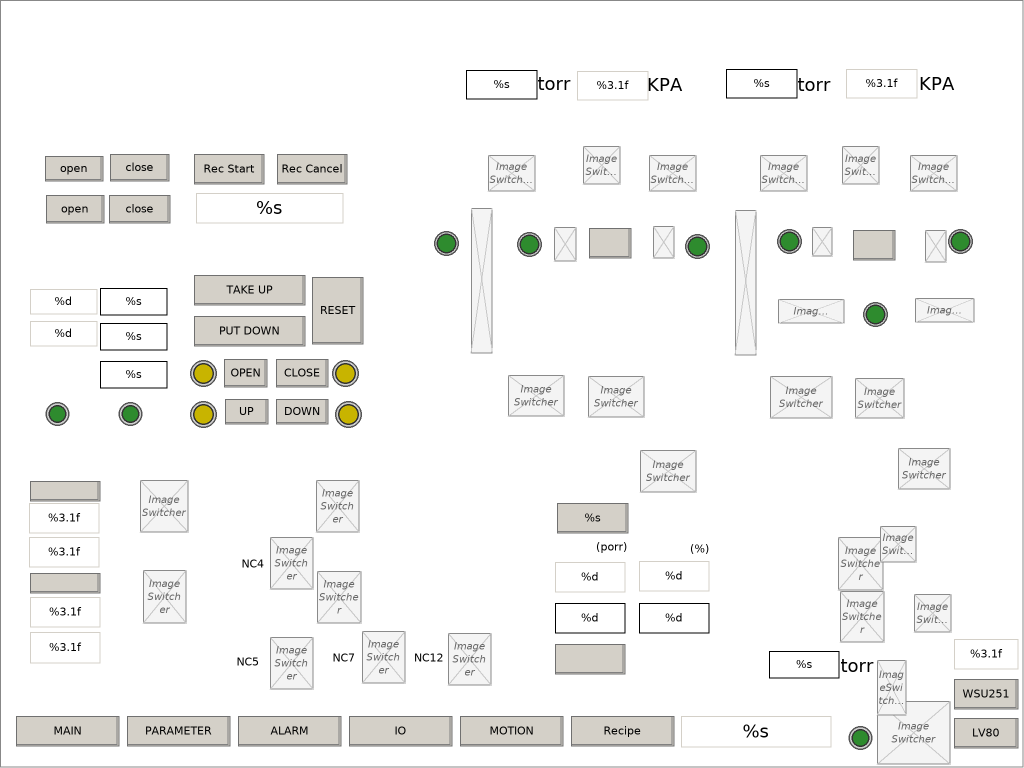
VISUALIZATION MainBase  // 1024x768, background image ImagePool_Base.LAYOUT
    ImageSwitcher (140,480 48x52), variable: DO2_0, background image: ImagePool_Base.VAL_ON, image: ImagePool_Base.VAL_OFF, behaviour: TOGGLE
    ImageSwitcher (143,570 43x53), variable: DO2_1, background image: ImagePool_Base.VAL_ON, image: ImagePool_Base.VAL_OFF, behaviour: TOGGLE
    ImageSwitcher (316,480 43x52), variable: DO2_2, background image: ImagePool_Base.VAL_ON, image: ImagePool_Base.VAL_OFF, behaviour: TOGGLE
    ImageSwitcher (317,571 44x52), variable: DO2_5, background image: ImagePool_Base.VAL_ON, image: ImagePool_Base.VAL_OFF, behaviour: TOGGLE
    ImageSwitcher (838,537 45x53), variable: DO4_0, background image: ImagePool_Base.VAL_ON, image: ImagePool_Base.VAL_OFF, behaviour: TOGGLE
    ImageSwitcher (649,155 47x36), variable: DO4_1, background image: ImagePool_Base.VAL_ON_RL, image: ImagePool_Base.VAL_OFF_RL, behaviour: TOGGLE
    ImageSwitcher (910,155 47x36), variable: DO4_2, background image: ImagePool_Base.VAL_ON_RL, image: ImagePool_Base.VAL_OFF_RL, behaviour: TOGGLE
    ImageSwitcher (840,591 44x51), variable: DO4_3, background image: ImagePool_Base.VAL_ON, image: ImagePool_Base.VAL_OFF, behaviour: TOGGLE
    ImageSwitcher (488,155 47x36), variable: DO4_4, background image: ImagePool_Base.VAL_ON_RL, image: ImagePool_Base.VAL_OFF_RL, behaviour: TOGGLE
    ImageSwitcher (760,155 47x36), variable: DO4_5, background image: ImagePool_Base.VAL_ON_RL, image: ImagePool_Base.VAL_OFF_RL, behaviour: TOGGLE
    ImageSwitcher (588,376 56x41), variable: DO2_7, background image: ImagePool_Base.VAL_ON_RL, image: ImagePool_Base.VAL_OFF_RL, behaviour: TOGGLE
    ImageSwitcher (508,375 56x41), variable: DO3_0, background image: ImagePool_Base.VAL_ON_RL, image: ImagePool_Base.VAL_OFF_RL, behaviour: TOGGLE
    ImageSwitcher (855,378 49x40), variable: DO3_1, background image: ImagePool_Base.VAL_ON_RL, image: ImagePool_Base.VAL_OFF_RL, behaviour: TOGGLE
    ImageSwitcher (770,376 62x42), variable: DO3_2, background image: ImagePool_Base.VAL_ON_RL, image: ImagePool_Base.VAL_OFF_RL, behaviour: TOGGLE
    ImageSwitcher (640,450 56x42), variable: DO4_7, background image: ImagePool_Base.VAL_ON_RL, image: ImagePool_Base.VAL_OFF_RL, behaviour: TOGGLE
    ImageSwitcher (898,448 52x41), variable: DO5_0, background image: ImagePool_Base.VAL_ON_RL, image: ImagePool_Base.VAL_OFF_RL, behaviour: TOGGLE
    ImageSwitcher (778,299 66x24), variable: DO5_6, background image: ImagePool_Base.HTR_ON, image: ImagePool_Base.HTR_OFF, behaviour: TOGGLE
    ImageSwitcher (915,298 59x24), variable: DO5_7, background image: ImagePool_Base.HTR_ON, image: ImagePool_Base.HTR_OFF, behaviour: TOGGLE
    Lamp1 (515,228 29x33), variable: MAIN.M2_SNR1, style: Lamp-Lamp1-Green
    Lamp1 (683,230 29x33), variable: MAIN.M2_SNR2, style: Lamp-Lamp1-Green
    Lamp1 (432,227 29x33), variable: MAIN.M1_sNR, style: Lamp-Lamp1-Green
    Lamp1 (946,225 29x33), variable: MAIN.M3_SNR2, style: Lamp-Lamp1-Green
    Lamp1 (775,225 29x33), variable: MAIN.M3_SNR1, style: Lamp-Lamp1-Green
    Lamp1 (861,298 29x33), variable: MAIN.M3_SNR3, style: Lamp-Lamp1-Green
    Rectangle (769,651 70x27), "%s", text variable: MAIN.show_CG1
    Rectangle (466,70 71x29), "%s", text variable: MAIN.show_CG2
    Rectangle (726,69 71x29), "%s", text variable: MAIN.show_CG3
    ImageSwitcher (653,226 21x32), variable: MOTION.LM_GoRight, input disabled if: MOTION.LM_GoLeft, background image: ImagePool_Base.RIGHT_ON, image: ImagePool_Base.RIGHT_OFF, behaviour: TOGGLE
    ImageSwitcher (812,227 20x29), variable: MOTION.RM_GoLeft, input disabled if: MOTION.RM_GoRight, background image: ImagePool_Base.LEFT_ON, image: ImagePool_Base.LEFT_OFF, behaviour: TOGGLE
    ImageSwitcher (925,230 21x32), variable: MOTION.RM_GoRight, input disabled if: MOTION.RM_GoLeft, background image: ImagePool_Base.RIGHT_ON, image: ImagePool_Base.RIGHT_OFF, behaviour: TOGGLE
    ImageSwitcher (554,227 22x34), variable: MOTION.LM_GoLeft, input disabled if: MOTION.LM_GoRight, background image: ImagePool_Base.LEFT_ON, image: ImagePool_Base.LEFT_OFF, behaviour: TOGGLE
    Textfield (577,71 71x29), "%3.1f", text variable: MAIN.ATM1_dis
    Textfield (846,69 71x29), "%3.1f", text variable: MAIN.ATM2_dis
    Textfield (954,639 64x30), "%3.1f", text variable: MAIN.ATM3_dis
    Textfield (29,503 70x30), "%3.1f", text variable: MAIN.MFC1_dis
    Textfield (30,597 70x30), "%3.1f", text variable: MAIN.MFC2_dis
    Textfield (29,537 70x30), "%3.1f", text variable: MFC1_Inp
        OnMouseClick: write the text variable via Default, min 0, max 1000
    Textfield (30,632 70x31), "%3.1f", text variable: MFC2_Inp
        OnMouseClick: write the text variable via Default, min 0, max 100
    Button (45,156 58x25), "open", input disabled if: GV1_OPN_DEVINP
        tap GV1_btn_open
    Button (110,154 59x27), "close", input disabled if: GV1_CLS_DEVINP
        tap GV1_btn_close
    Button (46,195 58x28), "open"
        tap GV2_btn_open
    Button (109,195 61x28), "close"
        tap GV2_btn_close
    ImageSwitcher (471,208 21x145), variable: DI2_1, background image: ImagePool_Base.GV_OPEN, image: ImagePool_Base.GV_CLS, behaviour: TOGGLE
    ImageSwitcher (735,210 21x145), variable: DI2_3, background image: ImagePool_Base.GV_OPEN, image: ImagePool_Base.GV_CLS, behaviour: TOGGLE
    Rectangle (100,288 67x27), "%s", text variable: MAIN.PV1
    Rectangle (100,323 67x27), "%s", text variable: MAIN.PV2
    Rectangle (100,361 67x27), "%s", text variable: MAIN.PV3
    Button (954,718 64x30), "LV80"
        toggle GVL.lv80_btn
    Button (954,679 64x30), "WSU251", input disabled if: MAIN.WSU_DEVINP
        toggle GVL.WSU_btn
    Lamp1 (847,722 27x32), variable: DI1_4, style: Lamp-Lamp1-Green
    Textfield (555,562 70x30), "%d", text variable: GVL.HTC_SetPr
        OnMouseClick: write the text variable via Default, min 0, max 300
    Textfield (639,561 70x30), "%d", text variable: GVL.HTC_SetPos
        OnMouseClick: write the text variable via Default, min 0, max 1000
    Rectangle (555,603 70x30), "%d", text variable: MAIN.HTC_ReadPr
    Rectangle (639,603 70x30), "%d", text variable: MAIN.HTC_ReadPos
    Button (555,644 70x30)
        toggle DO4_6
    Button (30,481 70x20)
        toggle mfc1_open_btn
    Button (30,573 70x20)
        toggle mfc2_open_btn
    Button (557,503 71x30), "%s", text variable: MAIN.cur_mode
        toggle MAIN.HTC_MODE_Pr
    Button (225,399 43x25), "UP"
        tap MAIN.m3_pin_up
    Button (276,399 52x25), "DOWN"
        tap MAIN.m3_pin_down
    Button (224,359 43x28), "OPEN"
        tap MAIN.m3_rail_open
    Button (276,359 52x28), "CLOSE"
        tap MAIN.M3_rail_CLOSE
    Lamp1 (188,355 31x37), variable: MAIN.M3_rail_opened, style: Lamp-Lamp1-Yellow
    Lamp1 (330,355 31x37), variable: MAIN.M3_rail_closed, style: Lamp-Lamp1-Yellow
    Lamp1 (188,396 31x37), variable: DI3_4, style: Lamp-Lamp1-Yellow
    Lamp1 (333,396 31x37), variable: DI3_5, style: Lamp-Lamp1-Yellow
    Textfield (30,289 67x25), "%d", text variable: GVL.SV1
        OnMouseClick: write the text variable via Default, min 0, max 300
    Textfield (30,321 67x25), "%d", text variable: GVL.SV2
        OnMouseClick: write the text variable via Default, min 0, max 300
    Button (194,275 111x30), "TAKE UP"
        tap MAIN.m3_up_btn
    Button (194,316 111x30), "PUT DOWN"
        tap MAIN.m3_down_btn
    ImageSwitcher (583,146 37x38), variable: MAIN.ATM1_STS, input disabled if: 1, background image: ImagePool_Base.ATM_ON, image: ImagePool_Base.ATM_OFF, behaviour: TOGGLE
    ImageSwitcher (842,146 37x38), variable: MAIN.ATM2_STS, input disabled if: 1, background image: ImagePool_Base.ATM_ON, image: ImagePool_Base.ATM_OFF, behaviour: TOGGLE
    ImageSwitcher (914,594 37x38), variable: MAIN.ATM3_STS, input disabled if: 1, background image: ImagePool_Base.ATM_ON, image: ImagePool_Base.ATM_OFF, behaviour: TOGGLE
    ImageSwitcher (877,701 73x63), variable: MAIN.LV80_STS, input disabled if: 1, background image: ImagePool_Base.LV80_ON, image: ImagePool_Base.LV80_OFF, behaviour: TOGGLE
    ImageSwitcher (877,660 29x55), variable: MAIN.WSU_STS, input disabled if: 1, background image: ImagePool_Base.WSU_ON, image: ImagePool_Base.WSU_OFF, behaviour: TOGGLE
    ImageSwitcher (880,526 36x36), variable: MAIN.TV_STS, input disabled if: 1, background image: ImagePool_Base.TV_ON, image: ImagePool_Base.TV_OFF, behaviour: TOGGLE
    Button (589,228 42x30)
        tap MOTION.LM_Stop
    Button (853,230 42x30)
        tap MOTION.RM_Stop
    Textfield (681,716 150x31), "%s", text variable: MAIN.cur_time
    Button (312,277 51x67), "RESET"
        tap MAIN.reset_btn
    Lamp1 (117,398 27x32), variable: DI1_6, style: Lamp-Lamp1-Green
    Lamp1 (44,398 27x32), variable: DI1_5, style: Lamp-Lamp1-Green
    Button (194,154 70x30), "Rec Start", colour toggle: GVL.Rec_start_btn
        toggle GVL.Rec_start_btn
    ImageSwitcher (270,537 43x52), variable: DO2_3, background image: ImagePool_Base.VAL_ON, image: ImagePool_Base.VAL_OFF, behaviour: TOGGLE
    ImageSwitcher (270,637 43x52), variable: DO2_4, background image: ImagePool_Base.VAL_ON, image: ImagePool_Base.VAL_OFF, behaviour: TOGGLE
    ImageSwitcher (362,631 43x52), variable: DO2_6, background image: ImagePool_Base.VAL_ON, image: ImagePool_Base.VAL_OFF, behaviour: TOGGLE
    ImageSwitcher (448,633 43x52), variable: DO3_3, background image: ImagePool_Base.VAL_ON, image: ImagePool_Base.VAL_OFF, behaviour: TOGGLE
    Label (532,69 44x30), "torr"
    Label (792,70 44x30), "torr"
    Label (233,549 40x30), "NC4"
    Label (228,647 40x30), "NC5"
    Label (324,643 40x30), "NC7"
    Label (409,643 40x30), "NC12"
    Label (835,651 44x30), "torr"
    Label (643,70 44x30), "KPA"
    Label (915,69 44x30), "KPA"
    Label (590,532 44x30), "(porr)"
    Label (678,534 44x30), "(%)"
    Button (16,716 103x30), "MAIN"
        OnMouseClick: change screen: MainBase
    Button (127,716 103x30), "PARAMETER"
        OnMouseClick: change screen: PARAMETER
    Button (238,716 103x30), "ALARM"
        OnMouseClick: change screen: ALARM
    Button (349,716 103x30), "IO"
        OnMouseClick: change screen: IO_TABLE
    Button (460,716 103x30), "MOTION"
        OnMouseClick: change screen: MOTION
    Button (571,716 103x30), "Recipe"
        OnMouseClick: change screen: Recipt
    Button (277,154 70x30), "Rec Cancel"
        tap Rec_stop_btn
    Textfield (196,193 147x30), "%s", text variable: GVL.CUR_step_name
END_VISUALIZATION

(* stored: Version 1.1.0.1, ProductVersion 3.1.4024.12
   Visu MainBase: Id {5d7fc6a1-2330-4deb-9294-64aba7aaa561} *)
